PROGRAM PRG_TEST
VAR
	fbMAV_DW_Test : FILTER_MAV_DW_Test; 
	fbMAV_W_Test : FILTER_MAV_W_Test; 
END_VAR

TcUnit.RUN();

END_PROGRAM

(* stored: Version 1.1.0.1, ProductVersion 3.1.4024.9
   POU PRG_TEST: Id {b6e50351-783e-4948-93d8-763e2dd52247}, SpecialFunc None *)
